{attribute 'qualified_only'}
{attribute 'strict'}
TYPE E_CabinetJob :
(
	Idle :=0,
	Initial,
	MoveIn,
	MoveOut,
	MovingOut,
	MovingIn,
	Moved,
	Finish,
	Error
);
END_TYPE

(* stored: Version 1.1.0.1, ProductVersion 3.1.4024.13
   DUT E_CabinetJob: Id {45000728-fc65-4a37-a123-2c12edc483f6} *)
